{attribute addProperty BoxType "EP2316-0008-0016"}
{attribute addProperty Id "InputAT %I*ARRAY[0 ..7] OF BOOL6480Sync_ErrorAT %I*BOOL8132"}
{attribute addProperty CRC "691952475"}
{attribute addProperty SizeInBites "72"}
{attribute addProperty SizeInBytes "9"}
TYPE DO_Inputs_9F71B9E2 :
STRUCT
	{attribute addProperty Name "Input"}
	Input AT %I* : ARRAY[0 ..7] OF BOOL;
	{attribute addProperty Name "Sync_Error"}
	Sync_Error AT %I* : BOOL;
END_STRUCT
END_TYPE

(* stored: Version 1.2.0.0, ProductVersion 3.1.4024.9
   DUT DO_Inputs_9F71B9E2: Id {1d0b374f-003d-4c3a-9104-e9190fa72279} *)
